// TIA Portal V20 export
VAR_GLOBAL   // PLC tag table "F-Digital_Inputs"
   FDI_EStopCh1 AT %I1000.0 : Bool;
   FDI_KeySettingModeCh1 AT %I1000.1 : Bool;
   FDI_KeySettingLaserCh1 AT %I1000.2 : Bool;
   FDI_EStopFeedback AT %I1000.3 : Bool;
   FDI_EStopCh2 AT %I1000.4 : Bool;
   FDI_KeySettingModeCh2 AT %I1000.5 : Bool;
   FDI_KeySettingLaserCh2 AT %I1000.6 : Bool;
   FDI_ExternalFeedback AT %I1000.7 : Bool;
   FDI_ReturnPowerLaser AT %I1008.0 : Bool;
   FDI_MaintenanceDoorClosedCh1 AT %I1008.1 : Bool;
   FDI_FrontDoorClosedCh1 AT %I1008.2 : Bool;
   FDI_EstopPowerLaserCh1 AT %I1008.3 : Bool;
   FDI_ReturnShutterLaser AT %I1008.4 : Bool;
   FDI_MaintenanceDoorClosedCh2 AT %I1008.5 : Bool;
   FDI_FrontDoorClosedCh2 AT %I1008.6 : Bool;
   FDI_EstopPowerLaserCh2 AT %I1008.7 : Bool;
   FDI_RoofLeftDoorClosedCh1 AT %I1016.0 : Bool;
   FDI_LaserKeyON_Ch1 AT %I1016.1 : Bool;
   FDI_LaserExternalDoorClosedCh1 AT %I1016.2 : Bool;
   FDI_IntOrExtSasGatesClosedCh1 AT %I1016.3 : Bool;
   FDI_RoofLeftDoorClosedCh2 AT %I1016.4 : Bool;
   FDI_LaserKeyON_Ch2 AT %I1016.5 : Bool;
   FDI_LaserExternalDoorClosedCh2 AT %I1016.6 : Bool;
   FDI_IntOrExtSasGatesClosedCh2 AT %I1016.7 : Bool;
   FDI_BW_LoaderDoorClosedCh1 AT %I1024.0 : Bool;
   FDI_RoofRightDoorClosedCh1 AT %I1024.1 : Bool;
   FDI_SonplasEstopCh1 AT %I1024.2 : Bool;
   FDI_BW_LoaderEStopCh1 AT %I1024.3 : Bool;
   FDI_BW_LoaderDoorClosedCh2 AT %I1024.4 : Bool;
   FDI_RoofRightDoorClosedCh2 AT %I1024.5 : Bool;
   FDI_SonplasEstopCh2 AT %I1024.6 : Bool;
   FDI_BW_LoaderEStopCh2 AT %I1024.7 : Bool;
   FDI_SonplasDoorClosedCh1 AT %I1032.0 : Bool;
   FDI_FreeI1032_1 AT %I1032.1 : Bool;
   FDI_FreeI1032_2 AT %I1032.2 : Bool;
   FDI_FreeI1032_3 AT %I1032.3 : Bool;
   FDI_SonplasDoorClosedCh2 AT %I1032.4 : Bool;
   FDI_FreeI1032_5 AT %I1032.5 : Bool;
   FDI_FreeI1032_6 AT %I1032.6 : Bool;
   FDI_DoorClosedFeedback AT %I1032.7 : Bool;
END_VAR
